ABB RobotStudio station: Lab4.rspag

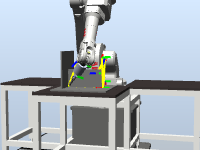
--- station ---
Station Lab4 (saved by RobotStudio 6.8.8307.1040)
Controller System1
  mechanical unit ROB_1: IRB1600_10_145__01, 6 joints, base frame (0, 0, 520) mm
Layout (positions relative to the parent item):
  - IRB1600_10_145__01 [mechanism, from Robots\IRB1600_10_145_G_01.rslib] at (0, 0, 520) mm; joint values [0.0527, 0.7066, 0.2561, -0.6317, 1.2328, 0] (rad or m)
  - Welding_case [part, from lab4\Welding_case.rslib] at (800, 0, 790) mm, rotated rx 0 ry 0 rz 90 deg
  - подставка [part, from System Volume Information\подставка.rslib]
  - rob-table [part, from System Volume Information\rob-table.rslib] at (218.5, 0, 0.5) mm
  - toolPencil [mechanism, from lab4\toolPencil.rslib] at (919.56, 12.21, 1000.49) mm, rotated rx -154.5 ry -38.42 rz -162.51 deg
Attachment: toolPencil is attached to IRB1600_10_145__01 / Link6
Targets, tools, work objects and paths stored in the station and not in the controller backup, written as RAPID:
! task T_ROB1
MODULE Module1
  CONST robtarget line_3_start:=[[218.5,327,0.5],[1,0,0,0],[0,-1,-1,0],[9E+09,9E+09,9E+09,9E+09,9E+09,9E+09]];
ENDMODULE


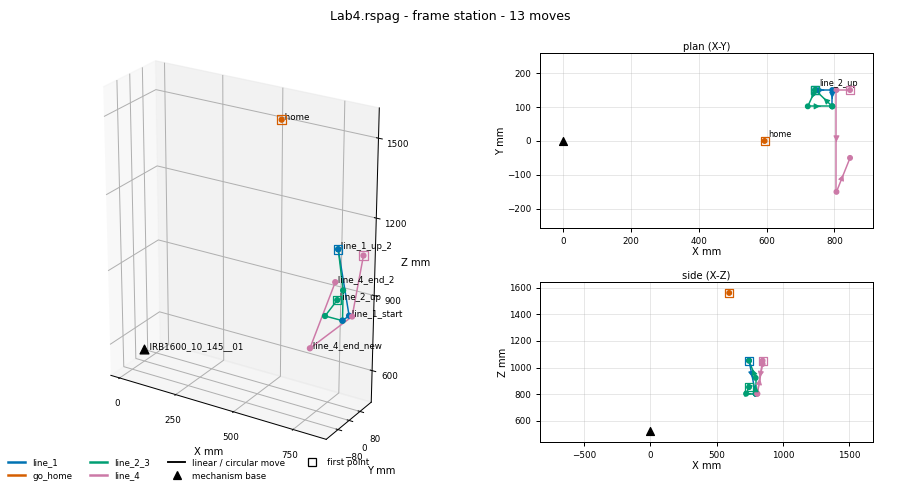
[picture p0: tool path of Lab4.rspag in frame station, 13 of 13 moves have a stored position in this frame; points joined in program order, loops and branches not executed]
--- Backups/System1/RAPID/TASK1/PROGMOD/CalibData.mod ---
MODULE CalibData
	PERS tooldata pen:=[TRUE,[[0,0,139],[1,0,0,0]],[0.5,[0,0,20],[1,0,0,0],0,0,0]];
	TASK PERS wobjdata wobjTable:=[FALSE,TRUE,"",[[348.622,-53.904,790],[1,0,0,0]],[[0,0,0],[1,0,0,0]]];
	TASK PERS wobjdata wobjWelding:=[FALSE,TRUE,"",[[575,-224.975,802],[1,0,0,0]],[[0,0,0],[1,0,0,0]]];
    PERS tooldata toolPencil:=[TRUE,[[0,0,280],[1,0,0,0]],[1,[0,0,1],[1,0,0,0],0,0,0]];
ENDMODULE

--- Backups/System1/RAPID/TASK1/PROGMOD/Module1.mod ---
MODULE Module1
	CONST robtarget line_1_up:=[[168.5,375,50],[0.382683432,0,0.923879533,0],[0,-1,-1,0],[9E+09,9E+09,9E+09,9E+09,9E+09,9E+09]];
	CONST robtarget line_1_start:=[[218.5,375,0.5],[0.382683432,0,0.923879533,0],[0,-2,1,0],[9E+09,9E+09,9E+09,9E+09,9E+09,9E+09]];
	CONST robtarget line_1_end:=[[218.5,327,0.5],[0.383022222,0.071497256,0.863069025,-0.321393805],[0,-2,1,0],[9E+09,9E+09,9E+09,9E+09,9E+09,9E+09]];
	CONST robtarget home:=[[594.25,0,1562.25],[0.382683432,0,0.923879533,0],[0,0,0,0],[9E+09,9E+09,9E+09,9E+09,9E+09,9E+09]];
	CONST robtarget line_1_up_2:=[[168.5,375,250],[0.382683432,0,0.923879533,0],[0,-2,1,0],[9E+09,9E+09,9E+09,9E+09,9E+09,9E+09]];
	CONST robtarget line_2_up:=[[168.5,375,50],[0.382683432,0,0.923879533,0],[0,-2,1,0],[9E+09,9E+09,9E+09,9E+09,9E+09,9E+09]];
	CONST robtarget line_2_start:=[[146.5,327,0.5],[0.300972014,0.247454494,0.800972014,-0.454561275],[0,-1,1,0],[9E+09,9E+09,9E+09,9E+09,9E+09,9E+09]];
	CONST robtarget line_2_end:=[[218.5,327,0.5],[0.37533331,0.104607774,0.831773471,-0.395392226],[0,-2,1,0],[9E+09,9E+09,9E+09,9E+09,9E+09,9E+09]];
	CONST robtarget line_3_end:=[[218.5,327,120],[0.653281482,0.27059805,0.653281482,-0.27059805],[0,-2,1,0],[9E+09,9E+09,9E+09,9E+09,9E+09,9E+09]];
    CONST robtarget line_4_up:=[[271,375,250],[0.258819045,0,-0.965925826,0],[0,-1,-1,0],[9E+09,9E+09,9E+09,9E+09,9E+09,9E+09]];
    CONST robtarget line_4_start:=[[231,375,0.5],[0.382683432,0,-0.923879533,0],[0,-1,-1,0],[9E+09,9E+09,9E+09,9E+09,9E+09,9E+09]];
    CONST robtarget line_4_end:=[[231,75,0.5],[0.115075127,-0.277815933,-0.881119571,0.364971676],[0,-1,-1,0],[9E+09,9E+09,9E+09,9E+09,9E+09,9E+09]];
    CONST robtarget line_4_end_2:=[[271,175,225],[0,0,0.923879533,-0.382683432],[0,-1,-1,0],[9E+09,9E+09,9E+09,9E+09,9E+09,9E+09]];
    CONST robtarget line_4_start_new:=[[230.999984738,374.999995266,0.500005537],[0.24476449,0.710193142,-0.590913792,-0.29417161],[0,0,-2,0],[9E+09,9E+09,9E+09,9E+09,9E+09,9E+09]];
    CONST robtarget line_4_end_new:=[[230.999994199,75.000006464,0.500012016],[0.285518991,0.211807221,-0.899272528,0.254804881],[0,-1,0,0],[9E+09,9E+09,9E+09,9E+09,9E+09,9E+09]];
    !***********************************************************
    !
    ! Module:  Module1
    !
    ! Description:
    !   <Insert description here>
    !
    ! Author: nikstol
    !
    ! Version: 1.0
    !
    !***********************************************************


    !***********************************************************
    !
    ! Procedure main
    !
    !   This is the entry point of your program
    !
    !***********************************************************
    PROC main()
		go_home;
		line_1;
		line_2_3;
		line_4;
		go_home;
        !Add your code here
    ENDPROC
	PROC line_1()
	    MoveL line_1_up_2,v50,fine,toolPencil\WObj:=wobjWelding;
	    MoveL line_1_start,v50,fine,toolPencil\WObj:=wobjWelding;
		MoveL line_1_end,v50,fine,toolPencil\WObj:=wobjWelding;
	ENDPROC
	PROC go_home()
	    MoveL home,v150,fine,pen\WObj:=wobj0;
	ENDPROC
	PROC line_2_3()
	    MoveL line_2_up,v50,fine,toolPencil\WObj:=wobjWelding;
	    MoveL line_2_start,v50,fine,toolPencil\WObj:=wobjWelding;
	    MoveL line_2_end,v50,fine,toolPencil\WObj:=wobjWelding;
	    MoveL line_3_end,v50,fine,toolPencil\WObj:=wobjWelding;
	    MoveL line_1_up_2,v50,fine,toolPencil\WObj:=wobjWelding;
	ENDPROC
    PROC line_4()
        MoveL line_4_up,v50,fine,toolPencil\WObj:=wobjWelding;
        MoveL line_4_start_new,v50,fine,toolPencil\WObj:=wobjWelding;
        MoveL line_4_end_new,v50,fine,toolPencil\WObj:=wobjWelding;
        MoveL line_4_end_2,v50,fine,toolPencil\WObj:=wobjWelding;
    ENDPROC
ENDMODULE
